// TIA Portal V19 program export: 0 tag tables, 0 data types, 1 data blocks, 2 code blocks (in call order from the OBs), 2 instance data blocks

DATA_BLOCK "Data_block_1"   // DB3
{ S7_Optimized_Access := 'TRUE' }
// stored: MemoryReserve 100
   VAR
      diStart : Bool;
      doDiode : Bool;
   END_VAR
BEGIN
END_DATA_BLOCK

ORGANIZATION_BLOCK "Main"   // OB1, LAD, ProgramCycle
TITLE = "Main Program Sweep (Cycle)"
{ S7_Optimized_Access := 'TRUE' }
// stored: SetENOAutomatically false
   VAR_INPUT
      Initial_Call : Bool;   // Initial call of this OB
      Remanence : Bool;   // =True, if remanent data are available
   END_VAR
BEGIN

REGION Network 1
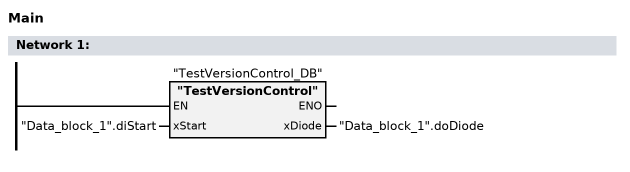
   RUNG wire#powerrail
      "TestVersionControl_DB"(xStart := "Data_block_1".diStart, xDiode => "Data_block_1".doDiode)
   END_RUNG
   // the same network as SCL:
   "TestVersionControl_DB"(xStart := "Data_block_1".diStart, xDiode => "Data_block_1".doDiode);   // "TestVersionControl"
END_REGION
END_ORGANIZATION_BLOCK

FUNCTION_BLOCK "TestVersionControl"
{ S7_Optimized_Access := 'TRUE' }
VERSION : 0.1
   VAR_INPUT 
      xStart : Bool;
   END_VAR

   VAR_OUTPUT 
      xDiode : Bool;
   END_VAR


BEGIN
	"R_TRIG_DB"(CLK := #xStart);
	
	
	IF "R_TRIG_DB".Q AND #xDiode = 0 THEN
	    #xDiode := 1;
	ELSIF "R_TRIG_DB".Q AND #xDiode = 1 THEN
	    #xDiode := 0;
	    ;
	END_IF;
	
	
END_FUNCTION_BLOCK

DATA_BLOCK "TestVersionControl_DB"   // DB2
// stored: InstanceOfName TestVersionControl, InstanceOfType FB
"TestVersionControl"
BEGIN
END_DATA_BLOCK

DATA_BLOCK "R_TRIG_DB"   // DB1
// stored: InstanceOfName R_TRIG, OfSystemLibElement R_TRIG, OfSystemLibVersion 1.0
"R_TRIG"
   // VAR_INPUT
   //    CLK : Bool;
   // END_VAR
   // VAR_OUTPUT
   //    Q : Bool;
   // END_VAR
   // VAR
   //    Stat_Bit : Bool;
   // END_VAR
BEGIN
END_DATA_BLOCK
